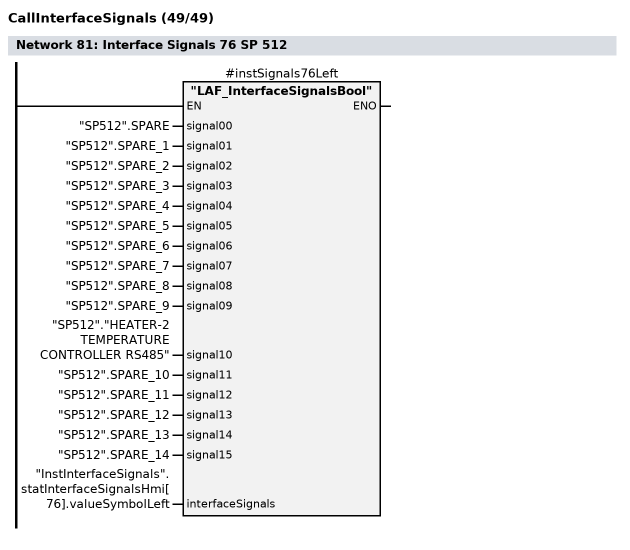
   RUNG wire#powerrail
      #instSignals76Left(signal00 := "SP512".SPARE, signal01 := "SP512".SPARE_1, signal02 := "SP512".SPARE_2, signal03 := "SP512".SPARE_3, signal04 := "SP512".SPARE_4, signal05 := "SP512".SPARE_5, signal06 := "SP512".SPARE_6, signal07 := "SP512".SPARE_7, signal08 := "SP512".SPARE_8, signal09 := "SP512".SPARE_9, signal10 := "SP512"."HEATER-2 TEMPERATURE CONTROLLER RS485", signal11 := "SP512".SPARE_10, signal12 := "SP512".SPARE_11, signal13 := "SP512".SPARE_12, signal14 := "SP512".SPARE_13, signal15 := "SP512".SPARE_14, interfaceSignals := "InstInterfaceSignals".statInterfaceSignalsHmi[76].valueSymbolLeft)
   END_RUNG
   // the same network as SCL:
   #instSignals76Left(signal00 := "SP512".SPARE,   // "LAF_InterfaceSignalsBool"
                      signal01 := "SP512".SPARE_1,
                      signal02 := "SP512".SPARE_2,
                      signal03 := "SP512".SPARE_3,
                      signal04 := "SP512".SPARE_4,
                      signal05 := "SP512".SPARE_5,
                      signal06 := "SP512".SPARE_6,
                      signal07 := "SP512".SPARE_7,
                      signal08 := "SP512".SPARE_8,
                      signal09 := "SP512".SPARE_9,
                      signal10 := "SP512"."HEATER-2 TEMPERATURE CONTROLLER RS485",
                      signal11 := "SP512".SPARE_10,
                      signal12 := "SP512".SPARE_11,
                      signal13 := "SP512".SPARE_12,
                      signal14 := "SP512".SPARE_13,
                      signal15 := "SP512".SPARE_14,
                      interfaceSignals := "InstInterfaceSignals".statInterfaceSignalsHmi[76].valueSymbolLeft);
END_REGION
END_FUNCTION_BLOCK
